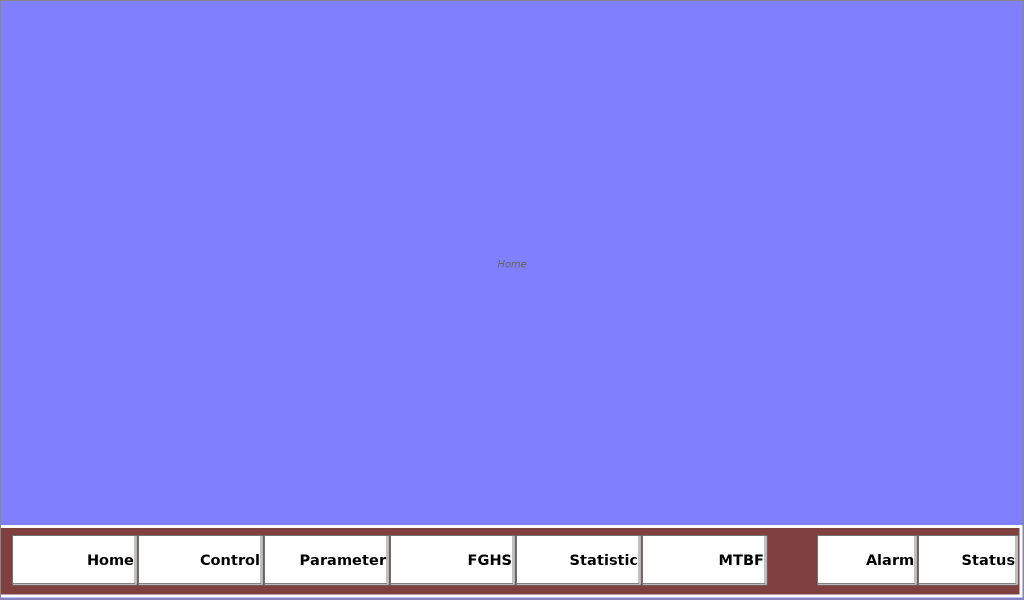
VISUALIZATION MainPage  // 1024x600
    Frame (0,0 1024x528)
        shows Home()
        shows Control()
        shows Parameter()
        shows FGHS()
        shows OEE()
        shows MTBF()
        shows Alarm()
        shows PLC_Status()
    Rectangle (-2,525 1024x72)
    Button (12,535 125x50), "Home", image: VisuSymbols.Symbols.Home
        OnMouseDown: FrameSelectionChange Selection=SelectedFrame=ea862550-edb1-43e7-b63a-bfe68bb940c3, GlobSel=AssignDir=MainPage.GenElemInst_1003, AssignType=Directly, SelType=Locally
    Button (138,535 125x50), "Control", image: VisuSymbols.Symbols.ControlPanel
        OnMouseDown: FrameSelectionChange Selection=SelectedFrame=ea862550-edb1-43e7-b63a-bfe68bb940c3, Selection=1, GlobSel=AssignType=Directly, SelType=Locally
    Button (817,535 100x50), "Alarm", image: VisuSymbols.Symbols.Caution
        OnMouseDown: FrameSelectionChange Selection=SelectedFrame=ea862550-edb1-43e7-b63a-bfe68bb940c3, Selection=6, GlobSel=AssignType=Directly, SelType=Locally
    Button (918,535 100x50), "Status", image: VisuSymbols.Symbols.Information
        OnMouseClick: FrameSelectionChange Selection=SelectedFrame=ea862550-edb1-43e7-b63a-bfe68bb940c3, Selection=7, GlobSel=AssignType=Directly, SelType=Locally
    Button (264,535 125x50), "Parameter", image: VisuSymbols.Symbols.TwoWheels
        OnMouseDown: FrameSelectionChange Selection=SelectedFrame=ea862550-edb1-43e7-b63a-bfe68bb940c3, Selection=2, GlobSel=AssignType=Directly, SelType=Locally
    Button (390,535 125x50), "FGHS", image: VisuSymbols.Symbols.Database
        OnMouseDown: FrameSelectionChange Selection=SelectedFrame=ea862550-edb1-43e7-b63a-bfe68bb940c3, Selection=3, GlobSel=AssignDir=MainPage.GenElemInst_1003, AssignType=Directly, SelType=Locally
    Button (516,535 125x50), "Statistic", image: VisuSymbols.Symbols.Diagram
        OnMouseDown: FrameSelectionChange Selection=SelectedFrame=ea862550-edb1-43e7-b63a-bfe68bb940c3, Selection=4, GlobSel=AssignDir=MainPage.GenElemInst_1003, AssignType=Directly, SelType=Locally
    Button (642,535 125x50), "MTBF", image: VisuSymbols.Symbols.Chart
        OnMouseDown: FrameSelectionChange Selection=SelectedFrame=ea862550-edb1-43e7-b63a-bfe68bb940c3, Selection=5, GlobSel=AssignDir=MainPage.GenElemInst_1003, AssignType=Directly, SelType=Locally
END_VISUALIZATION

(* stored: Version 1.1.0.1, ProductVersion 3.1.4024.12
   Visu MainPage: Id {b9e3df06-659e-4b55-8a3f-2de7ffe17db2} *)
